(* Logix 5000 project; controller Uidaho_Factory vendor 1 type 14 code 165 rev 38.11; software revision 38.00; part 3 of 3 *)
(* tags used below, declared in another part *)
   MPO_Done : BOOL;
   MPO_Turntable_Start : BOOL;
   Step : DINT[20];
   TurntableTimers : TIMER[10];
   PWM_Outputs : PWM_Out[20];
(* MainProgram, continued *)

ROUTINE MPO_Turntable_Process   (* ladder *)
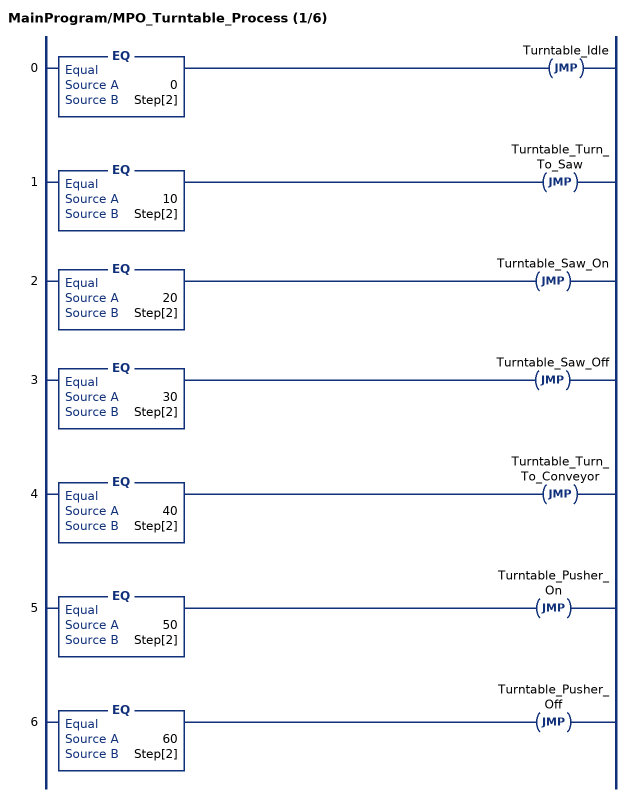
   0: EQ(0,Step[2])JMP(Turntable_Idle);
   1: EQ(10,Step[2])JMP(Turntable_Turn_To_Saw);
   2: EQ(20,Step[2])JMP(Turntable_Saw_On);
   3: EQ(30,Step[2])JMP(Turntable_Saw_Off);
   4: EQ(40,Step[2])JMP(Turntable_Turn_To_Conveyor);
   5: EQ(50,Step[2])JMP(Turntable_Pusher_On);
   6: EQ(60,Step[2])JMP(Turntable_Pusher_Off);
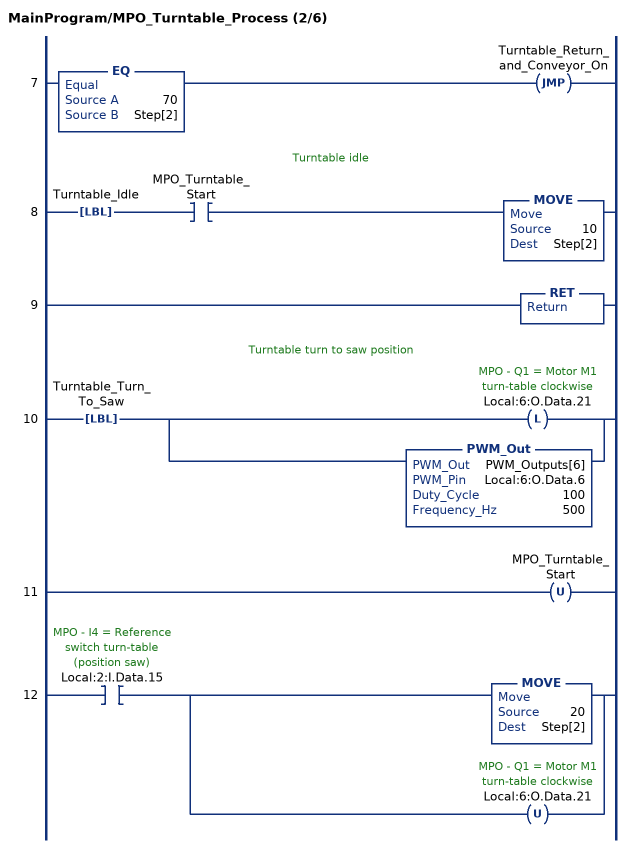
   7: EQ(70,Step[2])JMP(Turntable_Return_and_Conveyor_On);
   // Turntable idle
   8: LBL(Turntable_Idle)XIC(MPO_Turntable_Start)MOVE(10,Step[2]);
   9: RET();
   // Turntable turn to saw position
   10: LBL(Turntable_Turn_To_Saw)[OTL(Local:6:O.Data.21) ,PWM_Out(PWM_Outputs[6],Local:6:O.Data.6,100,500) ];
   11: OTU(MPO_Turntable_Start);
   12: XIC(Local:2:I.Data.15)[MOVE(20,Step[2]) ,OTU(Local:6:O.Data.21) ];
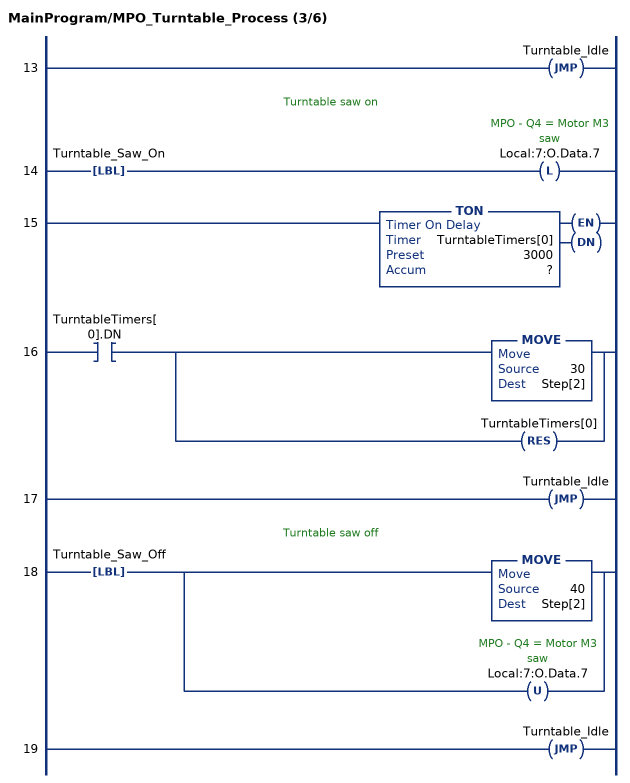
   13: JMP(Turntable_Idle);
   // Turntable saw on
   14: LBL(Turntable_Saw_On)OTL(Local:7:O.Data.7);
   15: TON(TurntableTimers[0],?,?);
   16: XIC(TurntableTimers[0].DN)[MOVE(30,Step[2]) ,RES(TurntableTimers[0]) ];
   17: JMP(Turntable_Idle);
   // Turntable saw off
   18: LBL(Turntable_Saw_Off)[MOVE(40,Step[2]) ,OTU(Local:7:O.Data.7) ];
   19: JMP(Turntable_Idle);
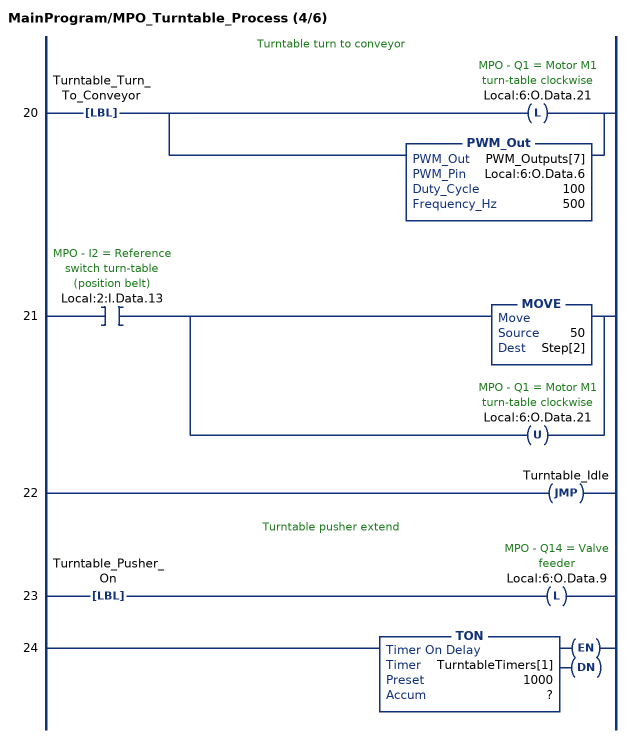
   // Turntable turn to conveyor
   20: LBL(Turntable_Turn_To_Conveyor)[OTL(Local:6:O.Data.21) ,PWM_Out(PWM_Outputs[7],Local:6:O.Data.6,100,500) ];
   21: XIC(Local:2:I.Data.13)[MOVE(50,Step[2]) ,OTU(Local:6:O.Data.21) ];
   22: JMP(Turntable_Idle);
   // Turntable pusher extend
   23: LBL(Turntable_Pusher_On)OTL(Local:6:O.Data.9);
   24: TON(TurntableTimers[1],?,?);
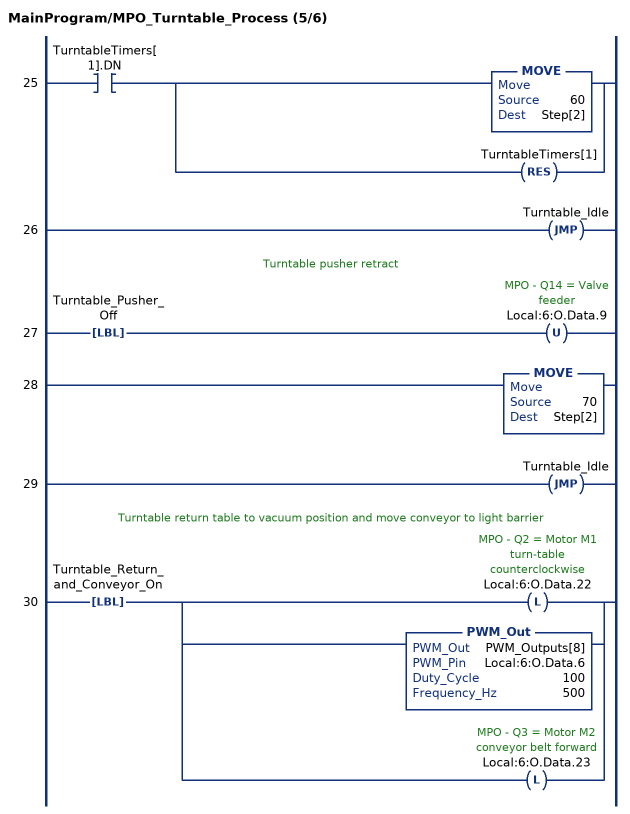
   25: XIC(TurntableTimers[1].DN)[MOVE(60,Step[2]) ,RES(TurntableTimers[1]) ];
   26: JMP(Turntable_Idle);
   // Turntable pusher retract
   27: LBL(Turntable_Pusher_Off)OTU(Local:6:O.Data.9);
   28: MOVE(70,Step[2]);
   29: JMP(Turntable_Idle);
   // Turntable return table to vacuum position and move conveyor to light barrier
   30: LBL(Turntable_Return_and_Conveyor_On)[[OTL(Local:6:O.Data.22) ,PWM_Out(PWM_Outputs[8],Local:6:O.Data.6,100,500) ] ,OTL(Local:6:O.Data.23) ];
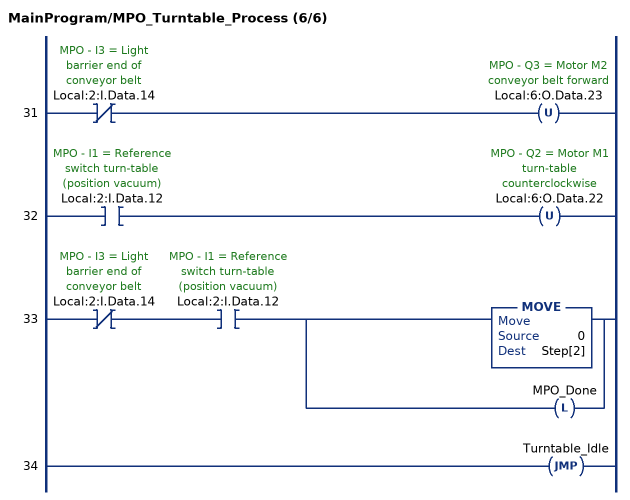
   31: XIO(Local:2:I.Data.14)OTU(Local:6:O.Data.23);
   32: XIC(Local:2:I.Data.12)OTU(Local:6:O.Data.22);
   33: XIO(Local:2:I.Data.14)XIC(Local:2:I.Data.12)[MOVE(0,Step[2]) ,OTL(MPO_Done) ];
   34: JMP(Turntable_Idle);
END_ROUTINE
END_PROGRAM
